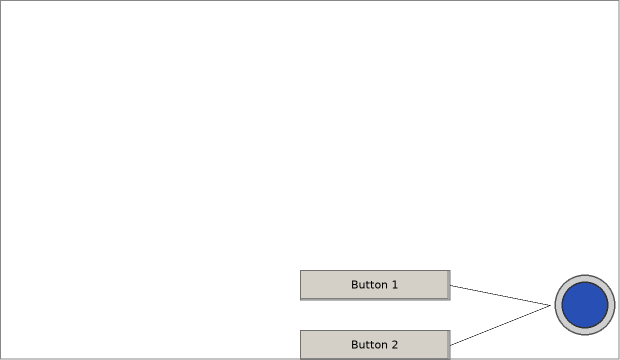
VISUALIZATION Visualization  // 620x360
    Button (300,270 150x30), "Button 1"
        OnMouseClick: toggle MAIN._Button1
    Button (300,330 150x30), "Button 2"
        OnMouseClick: toggle MAIN._Button2
    Lamp1 (550,270 70x70), variable: MAIN._Lamp, style: Lamp-Lamp1-Blue
    Line (450,285) (550,305)
    Line (450,345) (550,305)
END_VISUALIZATION

(* stored: Version 1.1.0.1
   Visu Visualization: Id {773dced3-3fad-4978-9d56-e700454a1d5a} *)
